FUNCTION_BLOCK Mode IMPLEMENTS I_Mode
VAR_INPUT
END_VAR
VAR_OUTPUT
END_VAR
VAR
	_mode : E_Mode;
END_VAR

PROPERTY Mode : E_Mode
GET
Mode := _mode;
END_GET
END_PROPERTY

END_FUNCTION_BLOCK

(* stored: Version 1.1.0.1
   POU Mode: Id {ea1b53db-cae0-4388-a4f6-e34f5637974b}, SpecialFunc None
   Property Mode: Id {41b0d16b-ab20-402a-a330-4395504f379d}
   Get Get: Id {b28bebd0-9c18-4f6f-95e1-4880ad08899e} *)
